LIN {X 0,Y 84.18,Z 344.932,A -85,B 0,C 180,E1 -31505.579,E2 -31505.579} C_VEL
LIN {X 0,Y 84.105,Z 345.156,A -85,B 0,C 180,E1 -31508.544,E2 -31508.544} C_VEL
LIN {X 0,Y 84.175,Z 345.975,A -85,B 0,C 180,E1 -31511.75,E2 -31511.75} C_VEL
LIN {X 0,Y 82.042,Z 358.989,A -85,B 0,C 180,E1 -31512.074,E2 -31512.074} C_VEL
LIN {X 0,Y 78.53,Z 371.76,A -85,B 0,C 180,E1 -31512.379,E2 -31512.379} C_VEL
LIN {X 0,Y 73.61,Z 384.422,A -85,B 0,C 180,E1 -31512.991,E2 -31512.991} C_VEL
LIN {X 0,Y 68.621,Z 394.241,A -85,B 0,C 180,E1 -31513.419,E2 -31513.419} C_VEL
LIN {X 0,Y 62.493,Z 404.055,A -85,B 0,C 180,E1 -31514.143,E2 -31514.143} C_VEL
LIN {X 0,Y 54.77,Z 414.177,A -85,B 0,C 180,E1 -31515.438,E2 -31515.438} C_VEL
LIN {X 0,Y 46.117,Z 423.367,A -85,B 0,C 180,E1 -31517.074,E2 -31517.074} C_VEL
LIN {X 0,Y 35.5,Z 432.535,A -85,B 0,C 180,E1 -31519.961,E2 -31519.961} C_VEL
LIN {X 0,Y 25.139,Z 439.78,A -85,B 0,C 180,E1 -31524.766,E2 -31524.766} C_VEL
LIN {X 0,Y 16.7,Z 444.681,A -85,B 0,C 180,E1 -31532.765,E2 -31532.765} C_VEL
LIN {X 0,Y 8.482,Z 448.948,A -85,B 0,C 180,E1 -31555.929,E2 -31555.929} C_VEL
LIN {X 0,Y 8.059,Z 453.156,A -85,B 0,C 180,E1 -31650.864,E2 -31650.864} C_VEL
LIN {X 0,Y 10.014,Z 453.798,A -85,B 0,C 180,E1 -31661.122,E2 -31661.122} C_VEL
LIN {X 0,Y 11.288,Z 455.737,A -85,B 0,C 180,E1 -31665.469,E2 -31665.469} C_VEL
LIN {X 0,Y 11.288,Z 600,A -85,B 0,C 180,E1 -31665.469,E2 -31665.469} C_VEL
LIN {X 0,Y 11.288,Z 600,A -85,B 0,C 180,E1 -31665.469,E2 -31665.469}

QRS_NEXT_CUT()

QRS_NEXT()
QRS_HOME()

END
